{attribute 'GeneratedUsingTerminal: IMecat-0007-0001'}
{attribute addProperty BoxType "IMecat-0007-0001"}
{attribute addProperty Id "Pdo_EntryAT %I*ARRAY[0..197] OF USINT198"}
{attribute addProperty CRC "1555868615"}
{attribute addProperty Size "198"}
TYPE DI_TxPDO_Map_16ADAB0E EXTENDS TcoIo.InputBase_8311D824 :
STRUCT
	{attribute addProperty Name "Pdo_Entry"}
	Pdo_Entry AT %I* : ARRAY[0..197] OF USINT;
END_STRUCT
END_TYPE

(* stored: Version 1.2.0.0, ProductVersion 3.1.4024.9
   DUT DI_TxPDO_Map_16ADAB0E: Id {6a1486bf-b75a-0d06-366a-a49de2b7a885} *)
